		M_ExeAction := pTarget^.M_CheckAction(refActionData, pMzTool); //Ausführbar mit Target?
		IF M_ExeAction > 0 THEN
			RETURN;
		END_IF
		
		M_ExeAction := pMzTool^.M_AskSiblingForAction(E_Action.ACTION_MoveToTarget);
		IF M_ExeAction > 0 THEN
			RETURN;
		END_IF
		
		
		eTargetRef := DINT_TO_USINT(refActionData.aParams[1]);
		nInsertLevel := DINT_TO_USINT(refActionData.aParams[4]);
		
		IF (pTarget^.P_eObjectGroup AND E_ObjectGroup.OBJECTGROUP_Rack) = E_ObjectGroup.OBJECTGROUP_Rack THEN
			pRack := pTarget;
			pPieceSlot := pRack^.M_GetSlot(DINT_TO_UINT(refActionData.aParams[2]));
		ELSIF pTarget^.P_eObjectType = E_ObjectType.OBJECTTYPE_Reactor THEN
			pReactor := pTarget;
			pPieceSlot := pReactor^.M_GetSlot(DINT_TO_UINT(refActionData.aParams[2]));
		ELSIF pTarget^.P_eObjectType = E_ObjectType.OBJECTTYPE_Mtp THEN
			pMtp := pTarget;
		END_IF
		
		IF eTargetRef = E_TargetRef.TARGETREF_Slot THEN
			IF pPieceSlot = 0 THEN
				M_ExeAction := E_ErrorIdCmd.ERRORID_InvalidTargetSlot;
				RETURN;
			ELSE
 				nTargetCol := UINT_TO_USINT(pPieceSlot^.nNr);
				nTargetRow := 0;
			END_IF
		ELSIF eTargetRef = E_TargetRef.TARGETREF_TwoDimArray THEN
			nTargetCol := DINT_TO_USINT(refActionData.aParams[2]);
			nTargetRow := DINT_TO_USINT(refActionData.aParams[3]);
		END_IF
	
	E_Action.ACTION_MeasureTool:
		bMeasureStamp := FALSE;
		bMeasureTarget := FALSE;
		bMeasureTip := FALSE;
		
		eMeasTipOption := DINT_TO_USINT(refActionData.aParams[2]);
		
		IF fbObjectDirectory.M_ObjIsTarget(refActionData.nTarget) THEN //Gültiges Target?
			pTarget := fbObjectDirectory.M_GetObjPointer(refActionData.nTarget);
		ELSE
			M_ExeAction := E_ErrorIdCmd.ERRORID_UnsuitableTarget;  //Error
			RETURN;
		END_IF		
	
		pMzTool := fbObjectDirectory.M_GetObjPointer(refActionData.nObject);
		IF pMzTool = 0 THEN
			M_ExeAction := E_ErrorIdCmd.ERRORID_ObjectNotExists;
			RETURN;
		END_IF
		
		CASE pMzTool^.P_eObjectType OF
			E_ObjectType.OBJECTTYPE_CartDispenser,
			E_ObjectType.OBJECTTYPE_CartDispStirrer,
			E_ObjectType.OBJECTTYPE_MultiCartHolder,
			E_ObjectType.OBJECTTYPE_PassivPip,
			E_ObjectType.OBJECTTYPE_PiezoPip,
			E_ObjectType.OBJECTTYPE_SolenoidPip,
			E_ObjectType.OBJECTTYPE_PowderPip,
			E_ObjectType.OBJECTTYPE_Extruder,
			E_ObjectType.OBJECTTYPE_TwinExtruder,
			E_ObjectType.OBJECTTYPE_Luer,
			E_ObjectType.OBJECTTYPE_TitrationTool,
			E_ObjectType.OBJECTTYPE_PickPlacePip:
				bMeasureTip := TRUE;
			E_ObjectType.OBJECTTYPE_HybridDispenser:
				//Gemessen wird mit dem MasterTool des Dispensers
				pHybridDispenser := pMzTool;
				pMzTool := pHybridDispenser^.P_pMasterTool;
				bMeasureTip := TRUE;
			E_ObjectType.OBJECTTYPE_StampSupport:	//Vermessung Stamp
				pStampSupport := fbObjectDirectory.M_GetObjPointer(refActionData.nObject);
				IF fbObjectDirectory.M_GetObjType(refActionData.nTarget) = E_ObjectType.OBJECTTYPE_InkStation THEN
					pInkStation := pTarget;
					iTargetZSensor := pInkStation^;
				ELSIF fbObjectDirectory.M_GetObjType(refActionData.nTarget) = E_ObjectType.OBJECTTYPE_StampMagazine THEN
					pStampMagazine := pTarget; 
					iTargetZSensor := pStampMagazine^;
				END_IF
				IF iTargetZSensor.P_bSensor THEN
					M_ExeAction := E_ErrorIdCmd.ERRORID_SensorAlreadySwitched;
					RETURN;
				END_IF
				bMeasureStamp := TRUE;
			E_ObjectType.OBJECTTYPE_ZSensor:	//Vermessung Target
				IF eMeasTipOption = E_MeasureOption.MEAS_OPTION_SlowApproach OR eMeasTipOption = E_MeasureOption.MEAS_OPTION_FastApproach THEN
					bMeasureTarget := TRUE;
				ELSE
					M_ExeAction := E_ErrorIdCmd.ERRORID_InvalidMeasureOption;
					RETURN;				
				END_IF
			ELSE
				M_ExeAction := E_ErrorIdCmd.ERRORID_UnsuitableObject; //Error
				RETURN;				
		END_CASE
		
		
		//Wenn bMeasureTip, dann muss Target ein TipCalibrator sein
		IF bMeasureTip OR bCalibrateTipCalibrator THEN
			IF NOT pTarget^.P_eObjectType = E_ObjectType.OBJECTTYPE_TipCalibrator THEN
				bMeasureTip := FALSE;
				bCalibrateTipCalibrator := FALSE;
				M_ExeAction := E_ErrorIdCmd.ERRORID_UnsuitableTarget;  //Error
				RETURN;
			END_IF
			pTipCalibrator := pTarget;
			bMeasureTipLegacy := pTipCalibrator^.P_bLegacy;
			
			IF pMzTool^.P_pPiece = 0 THEN
				IF pMzTool^.P_eObjectType = E_ObjectType.OBJECTTYPE_PassivPip OR
				   pMzTool^.P_eObjectType = E_ObjectType.OBJECTTYPE_PiezoPip OR
				   pMzTool^.P_eObjectType = E_ObjectType.OBJECTTYPE_SolenoidPip OR
				   pMzTool^.P_eObjectType = E_ObjectType.OBJECTTYPE_Luer THEN
				   rMeasureDistance := 6000;
				ELSIF pMzTool^.P_eObjectType = E_ObjectType.OBJECTTYPE_TitrationTool THEN 
				   rMeasureDistance := 10000;
				ELSE
					M_ExeAction := E_ErrorIdCmd.ERRORID_NoPieceOnTool;
					RETURN;
				END_IF
			ELSE
				IF NOT(pMzTool^.P_pPiece^.P_eObjectType = E_ObjectType.OBJECTTYPE_Nozzle OR
					pMzTool^.P_pPiece^.P_eObjectType = E_ObjectType.OBJECTTYPE_Needle OR
					pMzTool^.P_pPiece^.P_eObjectType = E_ObjectType.OBJECTTYPE_Tip) THEN
					M_ExeAction := E_ErrorIdCmd.ERRORID_InvalidPieceType;
					RETURN;
				ELSE
					rMeasureDistance := pMzTool^.P_pPiece^.P_rMeasureDistance;
				END_IF
			END_IF
		END_IF
		
		M_ExeAction := pMzTool^.M_CheckAction(refActionData, pTarget); //Action mit MzTool ausführbar?
		IF M_ExeAction > 0 THEN
			bMeasureTip := FALSE;
			RETURN;
		END_IF
		
		pHighVoltTray := pTarget^.M_GetFirstParentOfType(E_ObjectType.OBJECTTYPE_HighVoltTray);
		IF pHighVoltTray > 0 THEN
			IF pHighVoltTray^.P_nCurrentVoltage > cHighVoltThreshold THEN //>20 da anloger Eingang etwas rauscht
				M_ExeAction := E_ErrorIdCmd.ERRORID_RiskHighvoltFlashover;
				RETURN;
			END_IF
		END_IF
		
		
	E_Action.ACTION_MoveAllHome:
		;

	E_Action.ACTION_MoveToTarget:
		//Tool ermitteln
		IF fbObjectDirectory.M_ObjIsMzTool(refActionData.nObject) THEN //Gültiges MzTool?
			pMzTool := fbObjectDirectory.M_GetObjPointer(refActionData.nObject);
		ELSE 
			M_ExeAction := E_ErrorIdCmd.ERRORID_UnsuitableObject;  //Error
			RETURN;
		END_IF
		
		IF NOT (fbObjectDirectory.M_GetObjType(refActionData.nObject) = E_ObjectType.OBJECTTYPE_MZHead) THEN
			M_ExeAction := pMzTool^.M_AskSiblingForAction(E_Action.ACTION_MoveToTarget);
			IF M_ExeAction > 0 THEN
				RETURN;
			END_IF
		END_IF
		
		//Falls das Target sich auf dem HighVoltTray befindet und dieses auch angeschalten ist, dann ist ein MoveToTarget nur
		//mit einem MES-Tool möglich
		pTarget := fbObjectDirectory.M_GetObjPointer(refActionData.nTarget);
		IF pTarget = 0 THEN
			M_ExeAction := E_ErrorIdCmd.ERRORID_UnsuitableObject;  //Error
		END_IF
		pHighVoltTray := pTarget^.M_GetFirstParentOfType(E_ObjectType.OBJECTTYPE_HighVoltTray);
		IF pHighVoltTray > 0 THEN
			IF pHighVoltTray^.P_nCurrentVoltage > cHighVoltThreshold AND NOT pMzTool^.P_bIsMESTool THEN
				M_ExeAction := E_ErrorIdCmd.ERRORID_RiskHighvoltFlashover;
				RETURN;
			END_IF
		END_IF
	
		M_ExeAction := fbMoveToTarget.M_SetAndCheckParams(refActionData);

		IF M_ExeAction > 0 THEN
			RETURN;
		END_IF
		
	E_Action.ACTION_OpenCloseFlipTube:
		IF fbObjectDirectory.M_ObjIsMzTool(refActionData.nObject) THEN //Gültiges MzTool?
			pMzTool := fbObjectDirectory.M_GetObjPointer(refActionData.nObject);
		ELSE 
			M_ExeAction := E_ErrorIdCmd.ERRORID_UnsuitableObject;  //Error
			RETURN;
		END_IF
		
		IF fbObjectDirectory.M_ObjIsTarget(refActionData.nTarget) THEN //Gültiges Target?
			pTarget := fbObjectDirectory.M_GetObjPointer(refActionData.nTarget);
			IF pTarget^.P_eObjectType = E_ObjectType.OBJECTTYPE_FlipTubeRack THEN //Target ein FlipTubeRack?
				pFlipTubeRack := pTarget;
				pPieceSlot := pFlipTubeRack^.M_GetSlot(DINT_TO_UINT(refActionData.aParams[1]));
			ELSE
				M_ExeAction := E_ErrorIdCmd.ERRORID_UnsuitableTarget;  //Error	
			END_IF
		ELSE
			M_ExeAction := E_ErrorIdCmd.ERRORID_UnsuitableTarget;  //Error
			RETURN;
		END_IF
		
		M_ExeAction := pMzTool^.M_CheckAction(refActionData, pTarget); //Ausführbar mit Target?
		IF M_ExeAction > 0 THEN
			RETURN;
		END_IF
		
		M_ExeAction := pTarget^.M_CheckAction(refActionData, pMzTool); //Ausführbar mit MzTool?
		IF M_ExeAction > 0 THEN
			RETURN;
		END_IF
		bOpen := NOT DINT_TO_BOOL(refActionData.aParams[2]); //Öffen
		
	E_Action.ACTION_StampDemolding:
		IF fbObjectDirectory.M_GetObjType(refActionData.nObject) <> E_ObjectType.OBJECTTYPE_StampSupport THEN //Gültiges MzTool?
			M_ExeAction := E_ErrorIdCmd.ERRORID_UnsuitableObject;
			RETURN;
		END_IF
		pMzTool := fbObjectDirectory.M_GetObjPointer(refActionData.nObject);
		pStampSupport := pMzTool;

		M_ExeAction := pStampSupport^.M_CheckAction(refActionData,0);
		IF M_ExeAction > 0 THEN
			RETURN;
		END_IF
 
		nDistance1 := refActionData.aParams[1];
		nSpeed1 := refActionData.aParams[2];
		nPressure1 := DINT_TO_INT(refActionData.aParams[3]);
		nPressure2 := DINT_TO_INT(refActionData.aParams[4]);
		nPeriode := refActionData.aParams[5];
		nDutycycle := refActionData.aParams[6];
		
	E_Action.ACTION_StampInking:
		IF fbObjectDirectory.M_GetObjType(refActionData.nObject) <> E_ObjectType.OBJECTTYPE_StampSupport THEN //Gültiges MzTool?
			M_ExeAction := E_ErrorIdCmd.ERRORID_UnsuitableObject;
			RETURN;
		END_IF
		
		//Inking kann an einem Punkt oder an der InkStation stattfinden
		IF fbObjectDirectory.M_GetObjType(refActionData.nTarget) = E_ObjectType.OBJECTTYPE_InkStation THEN
			pInkStation := fbObjectDirectory.M_GetObjPointer(refActionData.nTarget);
		ELSIF fbObjectDirectory.M_GetObjType(refActionData.nTarget) = E_ObjectType.OBJECTTYPE_Point THEN
			pInkStation := 0;
		ELSE
			M_ExeAction := E_ErrorIdCmd.ERRORID_UnsuitableTarget;
			RETURN;
		END_IF
		
		//Wozu brauchen wir hier das Target?
		pTarget := fbObjectDirectory.M_GetObjPointer(refActionData.nTarget);
		pStampSupport := fbObjectDirectory.M_GetObjPointer(refActionData.nObject);
		
		M_ExeAction := pStampSupport^.M_CheckAction(refActionData,pTarget);
		IF M_ExeAction > 0 THEN
			RETURN;
		END_IF
		
		nDistance1 := refActionData.aParams[1];
		nPressure1 := DINT_TO_INT(refActionData.aParams[2]);
		nTime := DINT_TO_DWORD(refActionData.aParams[3]);
		
	E_Action.ACTION_TeachTarget:
		//Object gültig?
		IF NOT fbObjectDirectory.M_ObjIsMzTool(refActionData.nObject) THEN
			M_ExeAction := E_ErrorIdCmd.ERRORID_UnsuitableObject;  //Error
			RETURN;
		END_IF
		
		IF fbObjectDirectory.M_ObjIsTarget(refActionData.nTarget) THEN
			pTarget := fbObjectDirectory.M_GetObjPointer(refActionData.nTarget);
			IF pTarget > 0 THEN
				M_ExeAction := pTarget^.M_CheckAction(refActionData, pMzTool);
				IF M_ExeAction > 0 THEN
					RETURN;
				END_IF
			ELSE
				M_ExeAction := E_ErrorIdCmd.ERRORID_UnsuitableTarget;  //Error
				RETURN;
			END_IF
		ELSE
			M_ExeAction := E_ErrorIdCmd.ERRORID_UnsuitableTarget;  //Error
			RETURN;
		END_IF
		//Target gültig? (derzeit nur Mtp impl.)
		
		//Hier macht es Sinn, beim Target selber zu fragen, ob es sich einteachen lässt
		
		(*IF fbObjectDirectory.M_GetObjType(refActionData.nTarget) = E_ObjectType.OBJECTTYPE_Mtp THEN
			pMtp := aI_Object[refActionData.nTarget].P_pObject;
		ELSIF fbObjectDirectory.M_GetObjType(refActionData.nTarget) = E_ObjectType.OBJECTTYPE_Point THEN
			;
		ELSIF fbObjectDirectory.M_GetObjType(refActionData.nTarget) = E_ObjectType.OBJECTTYPE_Stroboscope THEN
			;
		ELSE
			M_ExeAction := E_ErrorIdCmd.ERRORID_InvalidTarget;  //Error
			RETURN;
		END_IF*)
		
		pMzTool := fbObjectDirectory.M_GetObjPointer(refActionData.nObject);
		pTarget := fbObjectDirectory.M_GetObjPointer(refActionData.nTarget);
		IF pTarget^.P_eObjectType = E_ObjectType.OBJECTTYPE_Mtp THEN
			pMtp := pTarget;
		END_IF
		eTargetRef := DINT_TO_USINT(refActionData.aParams[1]);
		nSpecPointSlotNr := DINT_TO_UINT(refActionData.aParams[2]);
		nZOffset1 := refActionData.aParams[3];
		//refActionData.aParams[4] ist Reserve
		eTeachOption := DINT_TO_USINT(refActionData.aParams[5]);
		
		pHighVoltTray := pTarget^.M_GetFirstParentOfType(E_ObjectType.OBJECTTYPE_HighVoltTray);
		IF pHighVoltTray > 0 THEN
			IF pHighVoltTray^.P_nCurrentVoltage > cHighVoltThreshold THEN
				M_ExeAction := E_ErrorIdCmd.ERRORID_RiskHighvoltFlashover;
				RETURN;
			END_IF
		END_IF
		
	E_Action.ACTION_TeachTool:
		IF NOT fbObjectDirectory.M_ObjIsMzTool(refActionData.nObject) THEN
			M_ExeAction := E_ErrorIdCmd.ERRORID_UnsuitableObject;  //Error
			RETURN;
		END_IF
		//Target gültig?
		IF NOT fbObjectDirectory.M_ObjIsTarget(refActionData.nTarget) THEN
			M_ExeAction := E_ErrorIdCmd.ERRORID_UnsuitableTarget;  //Error
			RETURN;
		END_IF
		pMzTool := fbObjectDirectory.M_GetObjPointer(refActionData.nObject);
		pTarget := fbObjectDirectory.M_GetObjPointer(refActionData.nTarget);
		eTargetRef := DINT_TO_USINT(refActionData.aParams[1]);
		nCol := DINT_TO_USINT(refActionData.aParams[2]);
		nRow := DINT_TO_USINT(refActionData.aParams[2]);
		nZOffset1 := refActionData.aParams[4];

		pHighVoltTray := pTarget^.M_GetFirstParentOfType(E_ObjectType.OBJECTTYPE_HighVoltTray);
		IF pHighVoltTray > 0 THEN
			IF pHighVoltTray^.P_nCurrentVoltage > cHighVoltThreshold THEN
				M_ExeAction := E_ErrorIdCmd.ERRORID_RiskHighvoltFlashover;
				RETURN;
			END_IF
		END_IF

	E_Action.ACTION_TransferGas:
		//Beteiligte Luers checken
		IF NOT fbObjectDirectory.M_GetObjType(refActionData.nObject) = E_ObjectType.OBJECTTYPE_Luer THEN
			M_ExeAction := E_ErrorIdCmd.ERRORID_UnsuitableObject;  //Error
			RETURN;
		END_IF

		IF NOT fbObjectDirectory.M_GetObjType(refActionData.nTarget) = E_ObjectType.OBJECTTYPE_Luer THEN
			M_ExeAction := E_ErrorIdCmd.ERRORID_UnsuitableObject;  //Error
			RETURN;
		END_IF
		pLuer := fbObjectDirectory.M_GetObjPointer(refActionData.nObject);
		pLuer2 := fbObjectDirectory.M_GetObjPointer(refActionData.nTarget);
		nPressure1 := DINT_TO_INT(refActionData.aParams[1]);
		nTime := DINT_TO_DWORD(refActionData.aParams[2]);
		
	E_Action.ACTION_TransferLiquid:
		//Beteiligte Luers checken
		IF NOT fbObjectDirectory.M_GetObjType(refActionData.nObject) = E_ObjectType.OBJECTTYPE_Luer THEN
			M_ExeAction := E_ErrorIdCmd.ERRORID_UnsuitableObject;  //Error
			RETURN;
		END_IF

		IF NOT fbObjectDirectory.M_GetObjType(refActionData.nTarget) = E_ObjectType.OBJECTTYPE_Luer THEN
			M_ExeAction := E_ErrorIdCmd.ERRORID_UnsuitableTarget;  //Error
			RETURN;
		END_IF
		pLuer := fbObjectDirectory.M_GetObjPointer(refActionData.nObject);
		pLuer2 := fbObjectDirectory.M_GetObjPointer(refActionData.nTarget);
		pDiluter1 := pLuer^.P_pDiluter;
		pDiluter2 := pLuer2^.P_pDiluter;
		
		nQuantity1 := refActionData.aParams[1];
		nFlow1 := refActionData.aParams[2];
		nQuantity2 := refActionData.aParams[3];
		nQuantity3 := refActionData.aParams[4];
		
	E_Action.ACTION_TransferTray:
		//Hier schon Bedingungen abfragen.
		IF fbObjectDirectory.M_GetObjType(refActionData.nObject) = E_ObjectType.OBJECTTYPE_TrayTransporter THEN
			pTrayTransporter := fbObjectDirectory.M_GetObjPointer(refActionData.nObject);
		ELSE
			M_ExeAction := E_ErrorIdCmd.ERRORID_UnsuitableObject;  //Error
			RETURN;
		END_IF
 
		eTransferTrayCtrl :=  DINT_TO_USINT(refActionData.aParams[1]);

	E_Action.ACTION_WashTool:
		IF fbObjectDirectory.M_ObjIsMzTool(refActionData.nObject) THEN //Gültiges MzTool?
			pMzTool := fbObjectDirectory.M_GetObjPointer(refActionData.nObject);
		ELSE 
			M_ExeAction := E_ErrorIdCmd.ERRORID_UnsuitableObject;  //Error
			RETURN;
		END_IF	
		
		IF fbObjectDirectory.M_GetObjType(refActionData.nTarget) <> E_ObjectType.OBJECTTYPE_WashStation THEN //gültiges Target?
			M_ExeAction := E_ErrorIdCmd.ERRORID_UnsuitableTarget;
			RETURN;
		ELSE
			pTarget := fbObjectDirectory.M_GetObjPointer(refActionData.nTarget);
			pWashStation := pTarget;
		END_IF
		
		//Kann Tool Action ausführen?
		M_ExeAction := pMzTool^.M_CheckAction(refActionData, pTarget);
		IF M_ExeAction > 0 THEN
			RETURN;
		END_IF
		
		//Kann WashStation Action ausführen?
		M_ExeAction := pWashStation^.M_CheckAction(refActionData, pMzTool);
		IF M_ExeAction > 0 THEN
			RETURN;
		END_IF
		
		nSpecPointSlotNr := DINT_TO_UINT(refActionData.aParams[1]);
		//RinseChannel aus WashStation holen
		nRinseChannel := pWashStation^.M_GetRinseChannel(UINT_TO_USINT(nSpecPointSlotNr));
		eWashMode := DINT_TO_USINT(refActionData.aParams[2]);
		//passt WashMode zu RinseChannel?
		IF (eWashMode = E_WashMode.MODE_WashInOutside) OR (eWashMode = E_WashMode.MODE_WashOutside) THEN
			IF nRinseChannel = 0 THEN
				M_ExeAction := E_ErrorIdCmd.ERRORID_InvalidRinseChannel;
				RETURN;
			END_IF
		END_IF
		
		nQuantity1 := refActionData.aParams[3];
		nFlow1 := refActionData.aParams[4];
		nTime := DINT_TO_DWORD(refActionData.aParams[5]);
		nDilInputNr := refActionData.aParams[6];

 	ELSE
		M_ExeAction := E_ErrorIdCmd.ERRORID_InvalidAction; //Error		
END_CASE
bBusy := TRUE;
eCurrentAction := refActionData.eAction;
eCurrentState := E_MachineState.MACHINESTATE_Active;
END_METHOD

METHOD M_Pause
VAR_INPUT
END_VAR
//derzeit wird nur DispenseTest in Pause versetzt
IF eCurrentState = E_MachineState.MACHINESTATE_Active THEN
	IF eCurrentAction = E_Action.ACTION_DispenseTest THEN
		eCurrentState := E_MachineState.MACHINESTATE_PauseRequest;
	END_IF
END_IF
END_METHOD

METHOD M_Reset
VAR_INPUT
END_VAR
VAR
END_VAR
IF eCurrentState = E_MachineState.MACHINESTATE_Error THEN
	bBusy := TRUE;
	eCurrentState := E_MachineState.MACHINESTATE_Reset;
END_IF
END_METHOD

METHOD M_Stop
VAR_INPUT
END_VAR
IF eCurrentState = E_MachineState.MACHINESTATE_Active OR 
	eCurrentState = E_MachineState.MACHINESTATE_PauseRequest OR
	eCurrentState = E_MachineState.MACHINESTATE_Pause THEN
	
	bStop := TRUE;
END_IF
END_METHOD

METHOD M_StopAction
VAR_INPUT
	eAction : E_Action;
END_VAR
IF eCurrentAction = eAction THEN
	M_Stop();
END_IF
END_METHOD

PROPERTY P_bLastActionResult : BOOL
GET
P_bLastActionResult := bLastActionResult;
END_GET
SET
bLastActionResult := P_bLastActionResult;
END_SET
END_PROPERTY

PROPERTY P_bPauseRequestIntern : BOOL
GET
P_bPauseRequestIntern := bPauseRequestIntern;
END_GET
SET
bPauseRequestIntern := P_bPauseRequestIntern;
END_SET
END_PROPERTY

PROPERTY P_nDispenseTrials : DINT
GET
P_nDispenseTrials := nDispenseTrials;
END_GET
SET
nDispenseTrials := P_nDispenseTrials;
END_SET
END_PROPERTY

PROPERTY P_nLastActionResult : DINT
GET
P_nLastActionResult := nLastActionResult;
END_GET
SET
nLastActionResult := P_nLastActionResult;
END_SET
END_PROPERTY

END_FUNCTION_BLOCK

(* stored: Version 1.1.0.1
   POU FB_ComplexAction: Id {b650c0e7-6803-4c22-baf8-46c779c7402e}, SpecialFunc None
   Action A_ActionOnArray: Id {81e29213-83c2-426b-b051-cdd527602f54}
   Action A_CalibrateTipCalibrator: Id {e30de4f8-4d0a-4bf8-82fb-c396f355d668}
   Action A_CalibrateZSensor: Id {eaa337a8-6f5a-4a5e-a875-8ba62a0cfd85}
   Action A_CleanTip: Id {916171ad-c85a-4b57-b6d1-fd3ca0193df7}
   Action A_CleanTipGen2: Id {5b08de20-f568-456c-9773-d9164f88616a}
   Action A_DispenseTest: Id {539f1f8e-f006-4a45-8a05-796e0e020375}
   Action A_DockTool: Id {61e0b189-07b1-41f9-8cc3-a58b3b542307}
   Action A_DryPip: Id {eeb51761-dba0-4a4f-ad48-db0b8d8778a9}
   Action A_DryToolInside: Id {ffce6e9a-aa96-407a-9004-3798e7509277}
   Action A_ExchangeNeedle: Id {2119df00-e3cf-42c0-89af-f1573b243765}
   Action A_ExchangepHCap: Id {d7125d14-3ca4-403b-a501-18a4f1ca4f89}
   Action A_ExchangeSeptum: Id {256d2556-f874-434e-b583-1e865fe9c0f6}
   Action A_ExchangeStamp: Id {5051ce3a-34cf-46cb-bcc4-f104e98da64a}
   Action A_ExchangeTip: Id {de90b719-326e-4176-9e18-63ba27c1803e}
   Action A_ExchangeVial: Id {2b5222c3-c230-4afc-a2e5-af790b6b06ef}
   Action A_ExchangeVialGripper: Id {be5abbc5-950d-46c0-8403-fff2b2635fe6}
   Action A_GetPipSample: Id {411b2e03-fc3b-4f77-9fa9-ac6299cd5cf1}
   Action A_InsertTool: Id {aedaf8f2-ada9-4e3f-863c-954f4394d794}
   Action A_MeasureStamp: Id {04a8f503-34af-4207-941e-bfa1bd861e3b}
   Action A_MeasureTarget: Id {65b22b02-811d-4b35-9f90-d8b418e4980f}
   Action A_MeasureTip: Id {330db07a-a078-4cb2-8c2e-d44f0a50b11b}
   Action A_MeasureTipLegacy: Id {94c78643-f9ab-41a2-957e-b5c06186e3a0}
   Action A_MoveAllHome: Id {09b08668-5879-4ea8-8541-958527d9d859}
   Action A_MoveToTarget: Id {c4de918c-5645-4b36-9ae8-fb7b00dc3998}
   Action A_OpenCloseFlipTube: Id {b1c54cc8-13da-44e7-ae11-bc442e1d2fe9}
   Action A_StampDemold: Id {45f90d75-d6c1-4e48-8331-193ecbc535b9}
   Action A_StampInking: Id {fd6b423a-c63a-4f65-a557-812b0863353e}
   Action A_TeachTarget: Id {29ae2d02-686f-4649-85a9-86f8d5314ceb}
   Action A_TeachTool: Id {58218c83-64a2-4f81-b5ac-78c2453db706}
   Action A_TransferGas: Id {a7bd9254-a499-40a9-8564-1e5eeacea37d}
   Action A_TransferLiquid: Id {9e1fa62f-48be-4177-8abb-ed228d3a5cff}
   Action A_TransferTray: Id {b4635470-f773-4dee-9ec0-01b2a106e557}
   Action A_TransferTrayLeftToSlot: Id {7c085589-7c41-4fab-8574-ac4ed088611f}
   Action A_TransferTrayRightToSlot: Id {fa6d4461-e4ef-4b76-a3f9-768d45e0fc29}
   Action A_TransferTraySlotToLeft: Id {478815e5-45ed-4b2a-962d-6dd2471a718a}
   Action A_TransferTraySlotToRight: Id {7f183d0b-1960-405a-90c8-be7941ebb145}
   Action A_WashTool: Id {e67038f0-0cd2-40d8-8fd9-6c024fecd1d8}
   Method FB_init: Id {a87249a9-16e6-4a89-8244-de38d471c1da}
   Method M_Continue: Id {06aa16b8-528c-4042-9e87-1adca7f253e9}
   Method M_ExeAction: Id {2dfbeeb4-beee-4d31-a41a-4d7e5517d911}
   Method M_Pause: Id {6563408b-852e-4c0f-ab85-e23e7f438d63}
   Method M_Reset: Id {79a03231-22de-4a6c-8a99-a05b6d451e8c}
   Method M_Stop: Id {d71e9176-0c8e-4c84-b35a-b8300efb494a}
   Method M_StopAction: Id {9d3a68bd-8a16-4853-9fed-0c9fe0b25844}
   Property P_bLastActionResult: Id {8ebef2e3-6fd7-4fca-b731-b24d0e9408e8}
   Get Get: Id {54fb2b42-db22-4810-8ac7-5cfda710b2a7}
   Set Set: Id {6275df5e-2354-496f-8529-b23dd9f0792a}
   Property P_bPauseRequestIntern: Id {0d9bc2f3-665b-4351-9efa-8db86a38487f}
   Get Get: Id {feb6accb-5185-4e09-81b6-1e45b3444f62}
   Set Set: Id {066cb2cd-0c53-4f6b-ae8f-8ed2b4f8aaa8}
   Property P_nDispenseTrials: Id {912744ba-1996-4cf0-9006-411438a1dbc4}
   Get Get: Id {6e4aa4a2-763f-43c6-9d65-e61fdc70c5d5}
   Set Set: Id {d134fbc9-0fa4-4628-acb8-e29270b81bbf}
   Property P_nLastActionResult: Id {3ab48b2d-f767-4878-8e53-d625bfa45943}
   Get Get: Id {bef90a69-1edc-46c7-aeb8-465533b7279b}
   Set Set: Id {68ba1c9e-b8af-4f0f-b0d7-f5334c22f0e6} *)
